Omron CX-Programmer project 新工程 (CX-Programmer 9.62)

# PLC JiBanYaHe: CP1L-E EM

## Global symbols (name address type ; comment)
ALM 0.04 BOOL  ; 轴1伺服报警
101.01 BOOL  ; 电磁阀2
1.05 BOOL  ; 光栅
1.06 BOOL  ; 退到位
1.07 BOOL  ; 进到位
200 CHANNEL  ; 减速
A643 CHANNEL  ; 压力当前值
D0 CHANNEL  ; 增速
D100 CHANNEL  ; 压力当前值
D102 CHANNEL  ; 当前位置
D2 CHANNEL  ; 脉冲数
D4 CHANNEL  ; 脉冲频率
H0 CHANNEL  ; 回原点速度
H12 CHANNEL  ; 保持时间
H2 CHANNEL  ; 原点坐标值
H4 CHANNEL  ; 上位
H6 CHANNEL  ; 快速
H8 CHANNEL  ; 慢速
W0.00 BOOL  ; 复位步
W0.01 BOOL  ; 等待启动步
W0.02 BOOL  ; 工作步
W0.03 BOOL  ; 等待取料完成
W10.00 BOOL  ; 电机驱动
W10.01 BOOL  ; 定位完成
W300.00 BOOL  ; 暂停
W50.00 BOOL  ; EMG Step
BEE 101.07 BOOL  ; 三色灯-蜂鸣器
DIR1 100.01 BOOL  ; 轴1（方向）
EMGB 1.03 BOOL  ; 急停【常闭】
FastLimit H10 WORD  ; 快压阀值
GREEN 101.06 BOOL  ; 三色灯-绿
NP 0.09 BOOL  ; 轴1反转极限【常闭】
PB 1.02 BOOL  ; 暂停
PLS1 100.00 BOOL  ; 轴1（脉冲）
PP 0.08 BOOL  ; 轴1正转极限【常闭】
RED 101.04 BOOL  ; 三色灯-红
RST 100.06 BOOL  ; 轴1伺服RST
SB1 1.00 BOOL  ; 启动1
SB2 1.01 BOOL  ; 启动2
SVN 100.04 BOOL  ; 轴1伺服ON
SlowLimit H11 WORD  ; 慢压阀值
VALVE 101.00 BOOL  ; 电磁阀1
VOCCUMV 1.04 BOOL  ; 负压表
YELLOW 101.05 BOOL  ; 三色灯-黄

## Program main (cyclic task 0)

### Section 段1

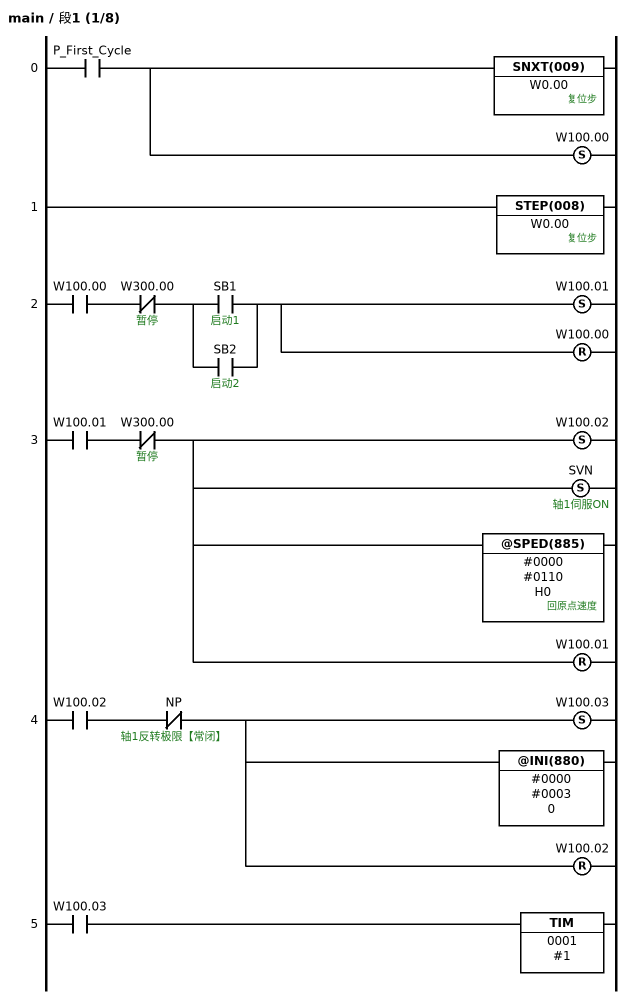
; rung 0
LD P_First_Cycle
SNXT(009) W0.00  ; 复位步
SET W100.00
; rung 1
STEP(008) W0.00  ; 复位步
; rung 2
LD W100.00
ANDNOT W300.00  ; 暂停
LD SB1  ; 启动1
OR SB2  ; 启动2
ANDLD
SET W100.01
RSET W100.00
; rung 3
LD W100.01
ANDNOT W300.00  ; 暂停
SET W100.02
SET SVN  ; 轴1伺服ON
@SPED(885) #0000 #0110 H0  ; 回原点速度
RSET W100.01
; rung 4
LD W100.02
ANDNOT NP  ; 轴1反转极限【常闭】
SET W100.03
@INI(880) #0000 #0003 0
RSET W100.02
; rung 5
LD W100.03
TIM 0001 #1

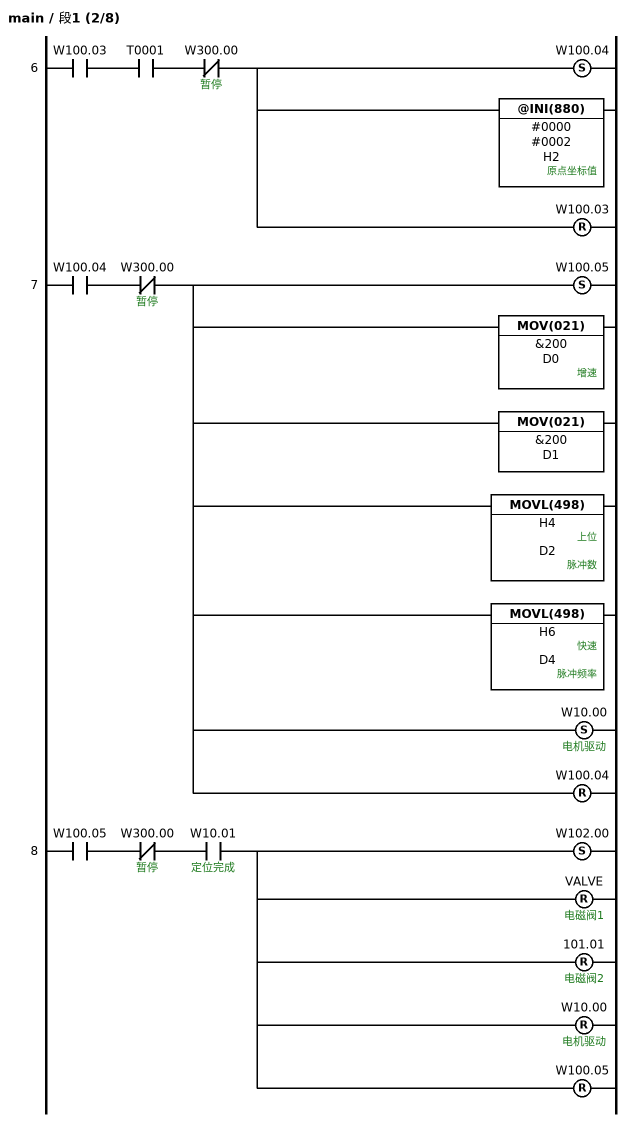
; rung 6
LD W100.03
AND T0001
ANDNOT W300.00  ; 暂停
SET W100.04
@INI(880) #0000 #0002 H2  ; 原点坐标值
RSET W100.03
; rung 7
LD W100.04
ANDNOT W300.00  ; 暂停
SET W100.05
MOV(021) &200 D0  ; 增速
MOV(021) &200 D1
MOVL(498) H4 D2  ; 上位, 脉冲数
MOVL(498) H6 D4  ; 快速, 脉冲频率
SET W10.00  ; 电机驱动
RSET W100.04
; rung 8
LD W100.05
ANDNOT W300.00  ; 暂停
AND W10.01  ; 定位完成
SET W102.00
RSET VALVE  ; 电磁阀1
RSET 101.01  ; 电磁阀2
RSET W10.00  ; 电机驱动
RSET W100.05

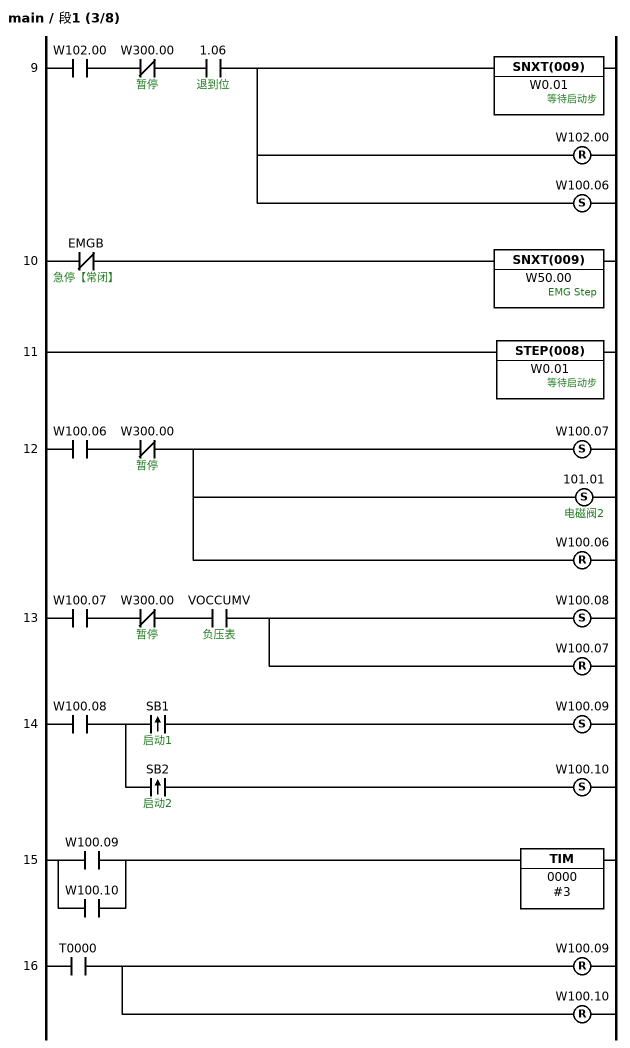
; rung 9
LD W102.00
ANDNOT W300.00  ; 暂停
AND 1.06  ; 退到位
SNXT(009) W0.01  ; 等待启动步
RSET W102.00
SET W100.06
; rung 10
LDNOT EMGB  ; 急停【常闭】
SNXT(009) W50.00  ; EMG Step
; rung 11
STEP(008) W0.01  ; 等待启动步
; rung 12
LD W100.06
ANDNOT W300.00  ; 暂停
SET W100.07
SET 101.01  ; 电磁阀2
RSET W100.06
; rung 13
LD W100.07
ANDNOT W300.00  ; 暂停
AND VOCCUMV  ; 负压表
SET W100.08
RSET W100.07
; rung 14
LD W100.08
OUT TR0
@AND SB1  ; 启动1
SET W100.09
LD TR0
@AND SB2  ; 启动2
SET W100.10
; rung 15
LD W100.09
OR W100.10
TIM 0000 #3
; rung 16
LD T0000
RSET W100.09
RSET W100.10

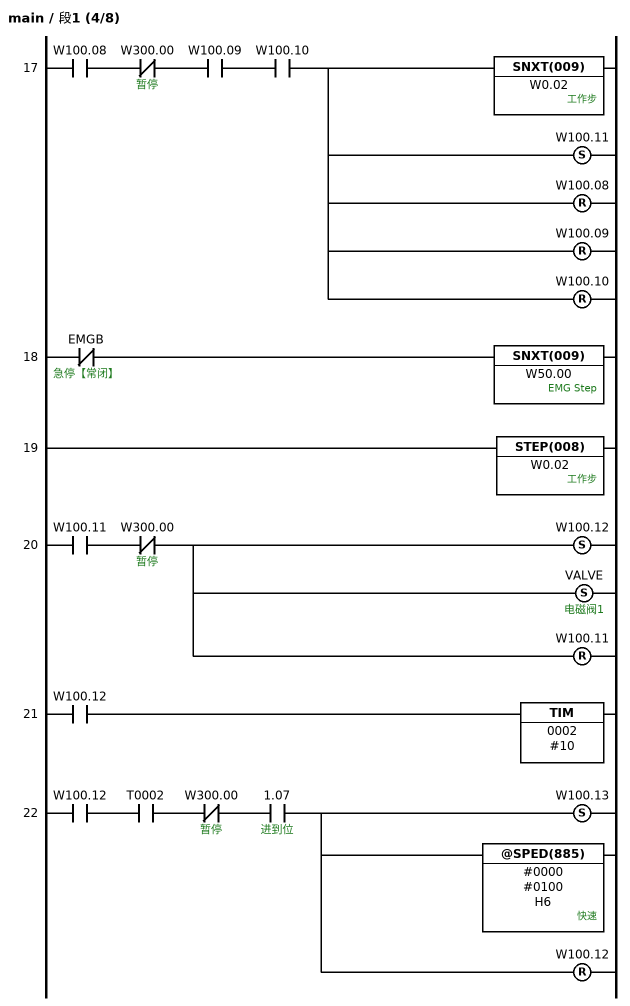
; rung 17
LD W100.08
ANDNOT W300.00  ; 暂停
AND W100.09
AND W100.10
SNXT(009) W0.02  ; 工作步
SET W100.11
RSET W100.08
RSET W100.09
RSET W100.10
; rung 18
LDNOT EMGB  ; 急停【常闭】
SNXT(009) W50.00  ; EMG Step
; rung 19
STEP(008) W0.02  ; 工作步
; rung 20
LD W100.11
ANDNOT W300.00  ; 暂停
SET W100.12
SET VALVE  ; 电磁阀1
RSET W100.11
; rung 21
LD W100.12
TIM 0002 #10
; rung 22
LD W100.12
AND T0002
ANDNOT W300.00  ; 暂停
AND 1.07  ; 进到位
SET W100.13
@SPED(885) #0000 #0100 H6  ; 快速
RSET W100.12

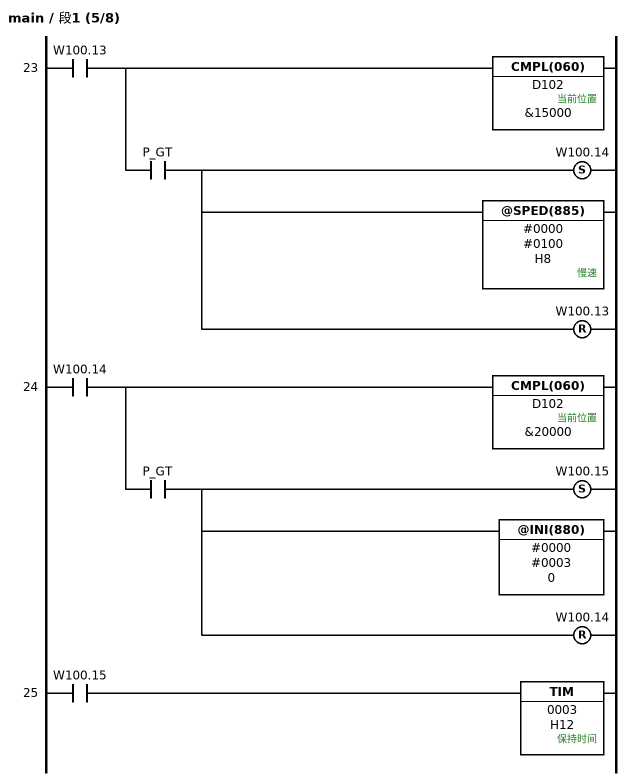
; rung 23
LD W100.13
CMPL(060) D102 &15000  ; 当前位置
AND P_GT
SET W100.14
@SPED(885) #0000 #0100 H8  ; 慢速
RSET W100.13
; rung 24
LD W100.14
CMPL(060) D102 &20000  ; 当前位置
AND P_GT
SET W100.15
@INI(880) #0000 #0003 0
RSET W100.14
; rung 25
LD W100.15
TIM 0003 H12  ; 保持时间

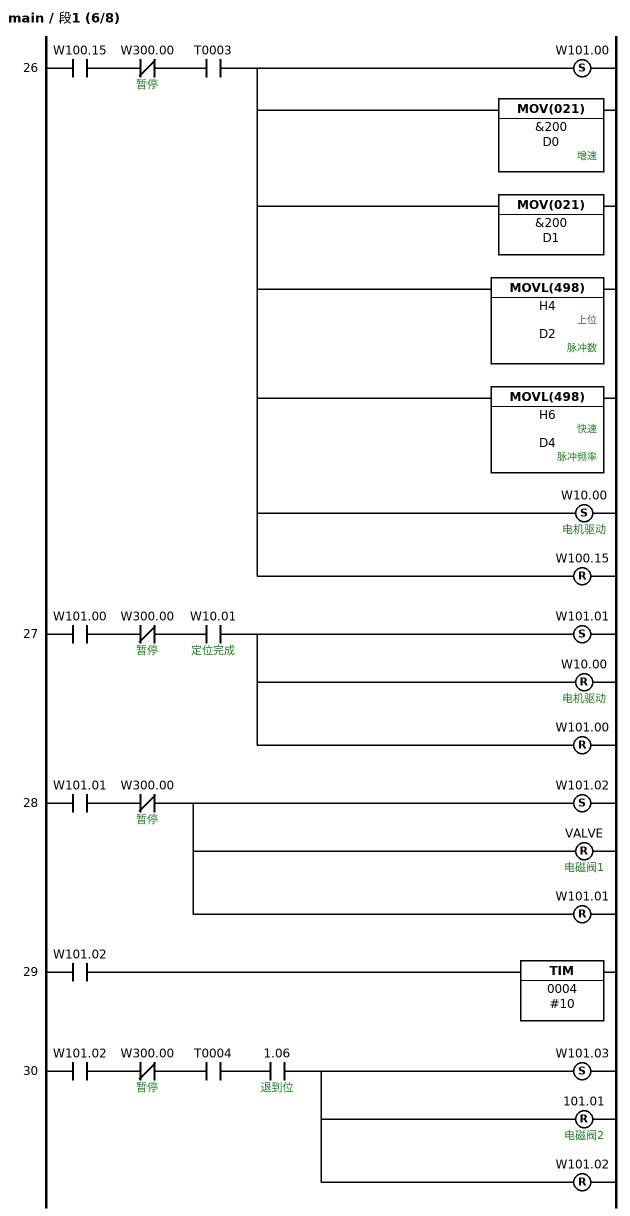
; rung 26
LD W100.15
ANDNOT W300.00  ; 暂停
AND T0003
SET W101.00
MOV(021) &200 D0  ; 增速
MOV(021) &200 D1
MOVL(498) H4 D2  ; 上位, 脉冲数
MOVL(498) H6 D4  ; 快速, 脉冲频率
SET W10.00  ; 电机驱动
RSET W100.15
; rung 27
LD W101.00
ANDNOT W300.00  ; 暂停
AND W10.01  ; 定位完成
SET W101.01
RSET W10.00  ; 电机驱动
RSET W101.00
; rung 28
LD W101.01
ANDNOT W300.00  ; 暂停
SET W101.02
RSET VALVE  ; 电磁阀1
RSET W101.01
; rung 29
LD W101.02
TIM 0004 #10
; rung 30
LD W101.02
ANDNOT W300.00  ; 暂停
AND T0004
AND 1.06  ; 退到位
SET W101.03
RSET 101.01  ; 电磁阀2
RSET W101.02

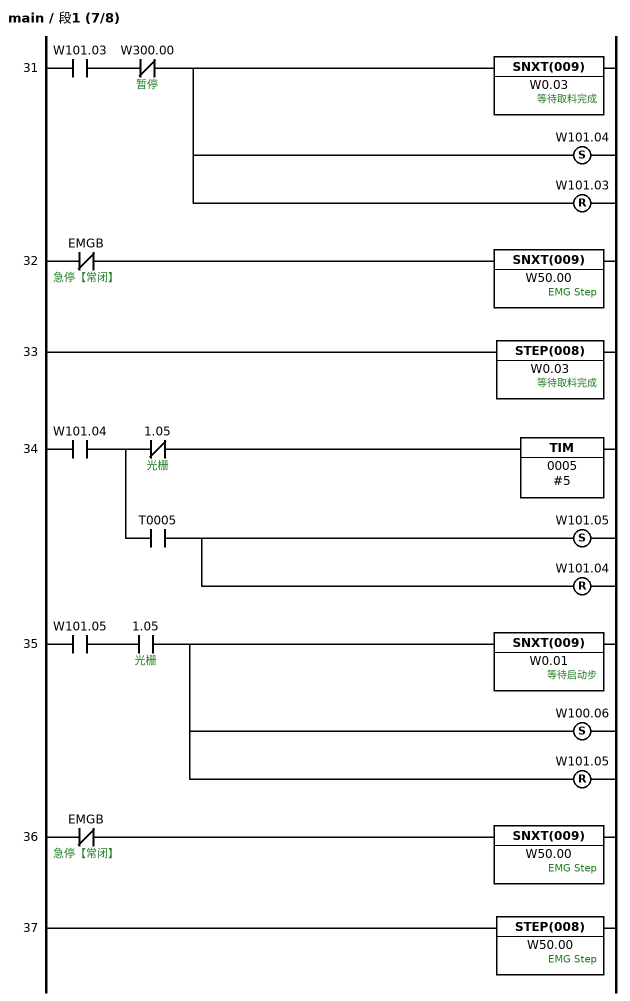
; rung 31
LD W101.03
ANDNOT W300.00  ; 暂停
SNXT(009) W0.03  ; 等待取料完成
SET W101.04
RSET W101.03
; rung 32
LDNOT EMGB  ; 急停【常闭】
SNXT(009) W50.00  ; EMG Step
; rung 33
STEP(008) W0.03  ; 等待取料完成
; rung 34
LD W101.04
OUT TR0
ANDNOT 1.05  ; 光栅
TIM 0005 #5
LD TR0
AND T0005
SET W101.05
RSET W101.04
; rung 35
LD W101.05
AND 1.05  ; 光栅
SNXT(009) W0.01  ; 等待启动步
SET W100.06
RSET W101.05
; rung 36
LDNOT EMGB  ; 急停【常闭】
SNXT(009) W50.00  ; EMG Step
; rung 37
STEP(008) W50.00  ; EMG Step

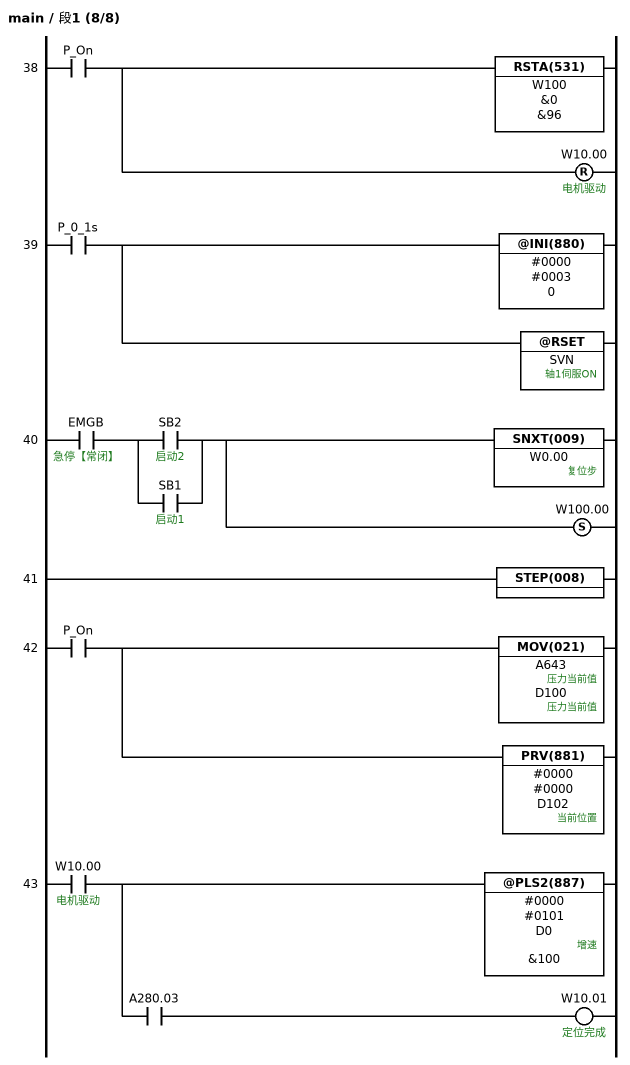
; rung 38
LD P_On
RSTA(531) W100 &0 &96
RSET W10.00  ; 电机驱动
; rung 39
LD P_0_1s
@INI(880) #0000 #0003 0
@RSET SVN  ; 轴1伺服ON
; rung 40
LD EMGB  ; 急停【常闭】
LD SB2  ; 启动2
OR SB1  ; 启动1
ANDLD
SNXT(009) W0.00  ; 复位步
SET W100.00
; rung 41
STEP(008)
; rung 42
LD P_On
MOV(021) A643 D100  ; 压力当前值
PRV(881) #0000 #0000 D102  ; 当前位置
; rung 43
LD W10.00  ; 电机驱动
@PLS2(887) #0000 #0101 D0 &100  ; 增速
AND A280.03
OUT W10.01  ; 定位完成

### Section END
; rung 0
END(001)